// TIA Portal V19 export
FUNCTION_BLOCK "A0304_Manager_FB"   // FB94, LAD
TITLE = Manager A0304
// stored: MemoryReserve 100, SetENOAutomatically false
   VAR_INPUT
      AreaInterface : "AreaInterface";
      ZSI : "udt_ZoneSafetyInterface";
      DataIn : Struct
         PbScaricaPacco : Bool;
         PbReggiaturaConclusa : Bool;
         LsMatPres1Load : Bool;
         LsMatPres2Load : Bool;
         LsMatPres1UnLoad : Bool;
         LsMatPres2UnLoad : Bool;
      END_STRUCT;
      CIn : Struct
         Navetta : Struct
            Testa : Struct
               Ax : "Positioning_DOL_Machine_COut";
               PalettiEsterni : "ValveMachine_COut";
               PalettiInterni : "ValveMachine_COut";
            END_STRUCT;
            Coda : Struct
               Ax : "Positioning_DOL_Machine_COut";
               PalettiEsterni : "ValveMachine_COut";
               PalettiInterni : "ValveMachine_COut";
            END_STRUCT;
            Cumulativo : Struct
               PalettiEsterni : "ValveMachine_COut";
               PalettiInterni : "ValveMachine_COut";
            END_STRUCT;
            ReadyToRecive : Bool;
         END_STRUCT;
         Sollevamento : Struct
            ReadyToDrop : Bool;   // In posizione di deposito e pacco completato
         END_STRUCT;
         Antiribaltamento : Struct
            Work : Bool;
            Rest : Bool;
            PalettoPos0 : Bool;
         END_STRUCT;
         Manager03 : Struct
            IsWaiting_NoPiecesBefore : Bool;
         END_STRUCT;
         ProdManager : "Prod_Beam_Ctrl";
      END_STRUCT;
   END_VAR
   VAR_OUTPUT
      COut { ExternalAccessible := 'False'; ExternalVisible := 'False'; ExternalWritable := 'False'} : Struct
         Navetta : Struct
            EnableStopDoorOpeningReq : Bool;
            EnableStopInPhase : Bool;
            EnableStopProgrammed : Bool;
            Control_ON : Bool;
            CanMoveFreely : Bool;
            OP : Struct
               VAI_A_PRELIEVO : Bool;
               PRELIEVO : Bool;
               VAI_A_DEPOSITO : Bool;
               DEPOSITO : Bool;
            END_STRUCT;
         END_STRUCT;
         Sollevatore : Struct
            ReadyToRecive : Bool;
            OutOfWorkspace : Bool;
         END_STRUCT;
      END_STRUCT;
      MachineInterface : "MachineInterface";
   END_VAR
   VAR_IN_OUT
      Par_Navetta : Struct
         PosPrePrelievo : LReal;
         PosPrelievo : LReal;
         PosDeposito : LReal;
         ToleranceWindow : LReal;
      END_STRUCT;
   END_VAR
   VAR
      Alarm : Struct
         ShuttleNotEmpty : Bool;
         STOP_FineTurno : Bool;
         STOP_ControlloQualita : Bool;
         STOP_End_Of_Proroduction : Bool;
         TimeoutRimozionePaccoMES : Bool;
      END_STRUCT;
      Warning : Struct
         UnloadNotPossible : Bool;   // impossibile scaricare con le porte aperte
         TimeoutRimozionePaccoMES : Bool;
      END_STRUCT;
      OP_CND : Struct
         VaiAPrelievo : Array[0..15] of "OpCnd";
         Prelievo { S7_SetPoint := 'True'} : Array[0..15] of "OpCnd";
         VaiADeposito : Array[0..15] of "OpCnd";
         Deposito : Array[0..15] of "OpCnd";
      END_STRUCT;
      Sts : Struct
         SemiAut : Struct
            ON : Bool;
            PbMaterialFwd : Bool;
            Request : Bool;
         END_STRUCT;
         InPosDeposito : Bool;
         InPosPrePrelievo : Bool;
         InPosPrelievo : Bool;
         RichiestaVaiDeposito : Bool;
         RichiestaVaiPrelievo : Bool;
         IsStandstill : Bool;
         AlarmsPresence : Bool;
         WarningsPresence : Bool;
      END_STRUCT;
      Ctrl : Struct
         Cycle : Struct
            VaiAPrelievo : Bool;   // CICLO - Vai a Posizione di prelievo
            Prelievo : Bool;   // CICLO - Prelievo
            VaiADeposito : Bool;   // CICLO - Vai a Posizione di deposito
            Deposito : Bool;   // CICLO - Deposito
         END_STRUCT;
         ReggiaturaConclusa : Bool;
         ConfermaPaccoScaricato : Bool;
         Stop : Bool;
      END_STRUCT;
      AUX : Struct
         SemiAut_Pb : Bool;
         PbScaricaPacco : Bool;
         PbReggiaturaConclusa : Bool;
      END_STRUCT;
      TON_MatPres : IEC_TIMER;
      TON_Stop : IEC_TIMER;
      TON_ForceConfermaPaccoScraicato : IEC_TIMER;
      TON_TimeoutRimozionePaccoMES { S7_SetPoint := 'True'} : IEC_TIMER;
      TON_WngTimeoutRimozionePaccoMES { S7_SetPoint := 'True'} : IEC_TIMER;
      CycleWithShortPiece : Bool;
   END_VAR
   VAR_TEMP
      PE : Struct
         PbScaricaPacco : Bool;
         PbReggiaturaConclusa : Bool;
      END_STRUCT;
      Testa_InPosDeposito : Bool;
      Testa_InPosPrePrelievo : Bool;
      Testa_InPosPrelievo : Bool;
      Coda_InPosDeposito : Bool;
      Coda_InPosPrePrelievo : Bool;
      Coda_InPosPrelievo : Bool;
      ConteggioLayer_Navetta : Int;
      i : Int;
   END_VAR
   VAR CONSTANT
      OUTOFWORKSPACE : LReal := 1000.0;   // Quota fuori ingombro navetta con sollevatore
   END_VAR
   VAR_TEMP   // added for the SCL form of the ladder/FBD networks
      _w1 : Bool;
      _w2 : Bool;
      _w3 : Bool;
      _w4 : Bool;
      _w5 : Bool;
   END_VAR
BEGIN

REGION Network 1 (SCL): Reset Alarms
   IF #AreaInterface.RstAlarms THEN
       #Alarm.ShuttleNotEmpty := FALSE;
       #Warning.UnloadNotPossible:=FALSE;
       #Alarm.STOP_ControlloQualita := FALSE;
       #Alarm.STOP_End_Of_Proroduction := FALSE;
       #Alarm.STOP_FineTurno := FALSE;
       #Alarm.TimeoutRimozionePaccoMES := FALSE;
   END_IF;
END_REGION

REGION Network 2: PE
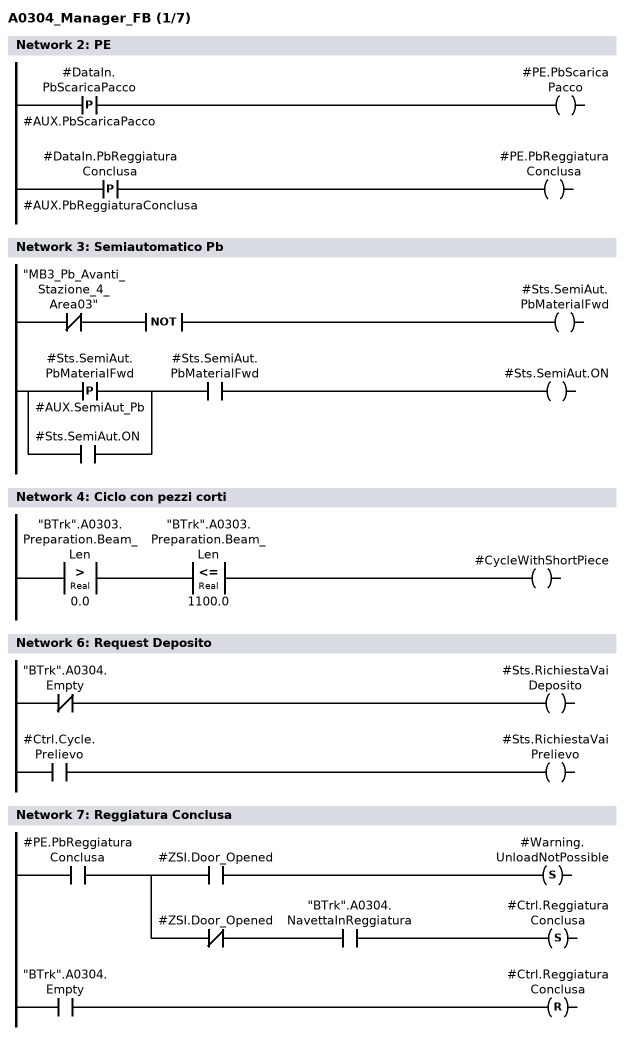
   RUNG wire#powerrail
      P_Contact(operand := #DataIn.PbScaricaPacco, bit := #AUX.PbScaricaPacco)
      Coil( #PE.PbScaricaPacco )
   END_RUNG
   RUNG wire#powerrail
      P_Contact(operand := #DataIn.PbReggiaturaConclusa, bit := #AUX.PbReggiaturaConclusa)
      Coil( #PE.PbReggiaturaConclusa )
   END_RUNG
   // the same network as SCL:
   #_w1 := #DataIn.PbScaricaPacco AND NOT #AUX.PbScaricaPacco;   // rising edge of #DataIn.PbScaricaPacco
   #AUX.PbScaricaPacco := #DataIn.PbScaricaPacco;
   #PE.PbScaricaPacco := #_w1;
   #_w2 := #DataIn.PbReggiaturaConclusa AND NOT #AUX.PbReggiaturaConclusa;   // rising edge of #DataIn.PbReggiaturaConclusa
   #AUX.PbReggiaturaConclusa := #DataIn.PbReggiaturaConclusa;
   #PE.PbReggiaturaConclusa := #_w2;
END_REGION

REGION Network 3: Semiautomatico Pb
   RUNG wire#powerrail
      I_Contact( "MB3_Pb_Avanti_Stazione_4_Area03" )
      Not()
      Coil( #Sts.SemiAut.PbMaterialFwd )
   END_RUNG
   RUNG wire#powerrail
      P_Contact(operand := #Sts.SemiAut.PbMaterialFwd, bit := #AUX.SemiAut_Pb)
      wire#w1
      Contact( #Sts.SemiAut.PbMaterialFwd )
      Coil( #Sts.SemiAut.ON )
   END_RUNG
   RUNG wire#powerrail
      Contact( #Sts.SemiAut.ON )
   END_RUNG wire#w1
   // the same network as SCL:
   #Sts.SemiAut.PbMaterialFwd := NOT (NOT "MB3_Pb_Avanti_Stazione_4_Area03");
   #_w1 := #Sts.SemiAut.PbMaterialFwd AND NOT #AUX.SemiAut_Pb;   // rising edge of #Sts.SemiAut.PbMaterialFwd
   #AUX.SemiAut_Pb := #Sts.SemiAut.PbMaterialFwd;
   #Sts.SemiAut.ON := (#_w1 OR #Sts.SemiAut.ON) AND #Sts.SemiAut.PbMaterialFwd;
END_REGION

REGION Network 4: Ciclo con pezzi corti
   RUNG wire#powerrail
      { S7_Templates := "SrcType := Real" } GT_Contact(in1 := "BTrk".A0303.Preparation.Beam_Len, in2 := 0.0)
      { S7_Templates := "SrcType := Real" } LE_Contact(in1 := "BTrk".A0303.Preparation.Beam_Len, in2 := 1100.0)
      Coil( #CycleWithShortPiece )
   END_RUNG
   // the same network as SCL:
   #CycleWithShortPiece := ("BTrk".A0303.Preparation.Beam_Len > 0.0) AND ("BTrk".A0303.Preparation.Beam_Len <= 1100.0);
END_REGION

REGION Network 6: Request Deposito
   RUNG wire#powerrail
      I_Contact( "BTrk".A0304.Empty )
      Coil( #Sts.RichiestaVaiDeposito )
   END_RUNG
   RUNG wire#powerrail
      Contact( #Ctrl.Cycle.Prelievo )
      Coil( #Sts.RichiestaVaiPrelievo )
   END_RUNG
   // the same network as SCL:
   #Sts.RichiestaVaiDeposito := NOT "BTrk".A0304.Empty;
   #Sts.RichiestaVaiPrelievo := #Ctrl.Cycle.Prelievo;
END_REGION

REGION Network 7: Reggiatura Conclusa
   RUNG wire#powerrail
      Contact( #PE.PbReggiaturaConclusa )
      wire#w1
      Contact( #ZSI.Door_Opened )
      S_Coil( #Warning.UnloadNotPossible )
   END_RUNG
   RUNG wire#w1
      I_Contact( #ZSI.Door_Opened )
      Contact( "BTrk".A0304.NavettaInReggiatura )
      S_Coil( #Ctrl.ReggiaturaConclusa )
   END_RUNG
   RUNG wire#powerrail
      Contact( "BTrk".A0304.Empty )
      R_Coil( #Ctrl.ReggiaturaConclusa )
   END_RUNG
   // the same network as SCL:
   IF #PE.PbReggiaturaConclusa AND #ZSI.Door_Opened THEN #Warning.UnloadNotPossible := TRUE; END_IF;
   IF #PE.PbReggiaturaConclusa AND NOT #ZSI.Door_Opened AND "BTrk".A0304.NavettaInReggiatura THEN
       #Ctrl.ReggiaturaConclusa := TRUE;
   END_IF;
   IF "BTrk".A0304.Empty THEN #Ctrl.ReggiaturaConclusa := FALSE; END_IF;
END_REGION

REGION Network 8: Conferma Pacco Scaricato
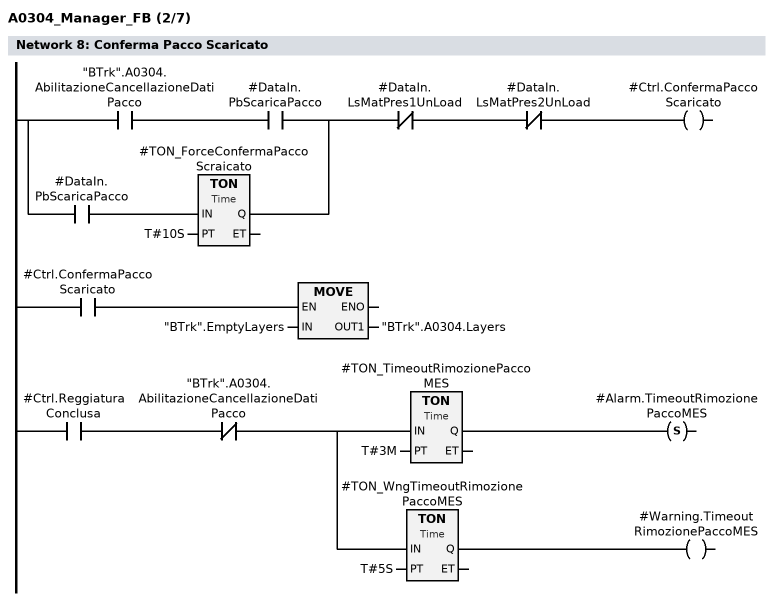
   RUNG wire#powerrail
      Contact( "BTrk".A0304.AbilitazioneCancellazioneDatiPacco )
      Contact( #DataIn.PbScaricaPacco )
      wire#w1
      I_Contact( #DataIn.LsMatPres1UnLoad )
      I_Contact( #DataIn.LsMatPres2UnLoad )
      Coil( #Ctrl.ConfermaPaccoScaricato )
   END_RUNG
   RUNG wire#powerrail
      Contact( #DataIn.PbScaricaPacco )
      { S7_Templates := "time_type := Time" } #TON_ForceConfermaPaccoScraicato.TON(pt := T#10S, et =>)
   END_RUNG wire#w1
   RUNG wire#powerrail
      Contact( #Ctrl.ConfermaPaccoScaricato )
      Move(in := "BTrk".EmptyLayers, out1 => "BTrk".A0304.Layers)
   END_RUNG
   RUNG wire#powerrail
      Contact( #Ctrl.ReggiaturaConclusa )
      I_Contact( "BTrk".A0304.AbilitazioneCancellazioneDatiPacco )
      wire#w2
      { S7_Templates := "time_type := Time" } #TON_TimeoutRimozionePaccoMES.TON(pt := T#3M, et =>)
      S_Coil( #Alarm.TimeoutRimozionePaccoMES )
   END_RUNG
   RUNG wire#w2
      { S7_Templates := "time_type := Time" } #TON_WngTimeoutRimozionePaccoMES.TON(pt := T#5S, et =>)
      Coil( #Warning.TimeoutRimozionePaccoMES )
   END_RUNG
   // the same network as SCL:
   #TON_ForceConfermaPaccoScraicato.TON(IN := #DataIn.PbScaricaPacco, PT := T#10S);
   #Ctrl.ConfermaPaccoScaricato := (("BTrk".A0304.AbilitazioneCancellazioneDatiPacco AND #DataIn.PbScaricaPacco) OR #TON_ForceConfermaPaccoScraicato.Q) AND NOT #DataIn.LsMatPres1UnLoad AND NOT #DataIn.LsMatPres2UnLoad;
   IF #Ctrl.ConfermaPaccoScaricato THEN "BTrk".A0304.Layers := "BTrk".EmptyLayers; END_IF;
   #_w1 := #Ctrl.ReggiaturaConclusa AND NOT "BTrk".A0304.AbilitazioneCancellazioneDatiPacco;
   #TON_TimeoutRimozionePaccoMES.TON(IN := #_w1, PT := T#3M);
   IF #TON_TimeoutRimozionePaccoMES.Q THEN #Alarm.TimeoutRimozionePaccoMES := TRUE; END_IF;
   #TON_WngTimeoutRimozionePaccoMES.TON(IN := #_w1, PT := T#5S);
   #Warning.TimeoutRimozionePaccoMES := #TON_WngTimeoutRimozionePaccoMES.Q;
END_REGION

REGION Network 10: Ax Navetta in posizione
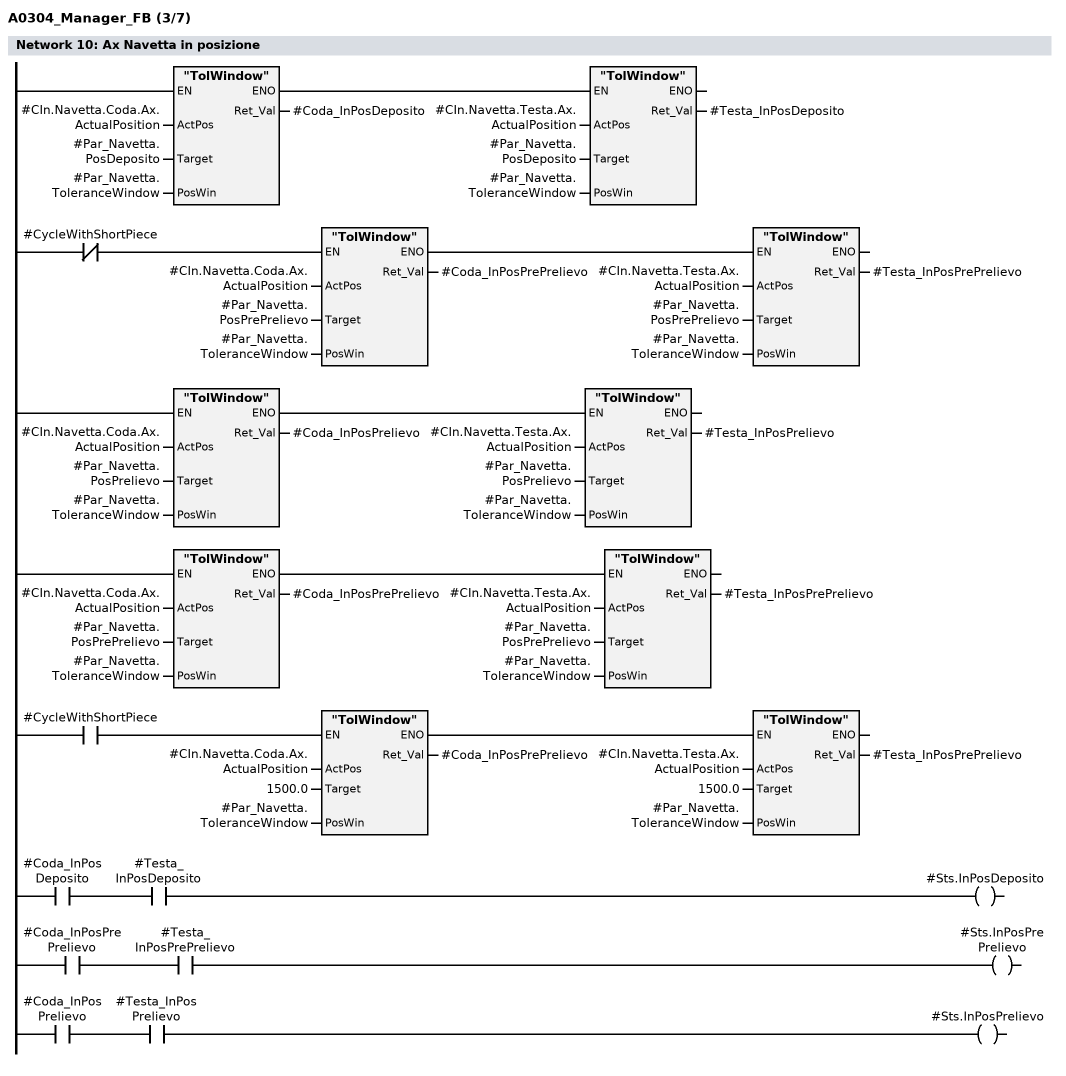
   RUNG wire#powerrail
      "TolWindow"(ActPos := #CIn.Navetta.Coda.Ax.ActualPosition, Target := #Par_Navetta.PosDeposito, PosWin := #Par_Navetta.ToleranceWindow, Ret_Val => #Coda_InPosDeposito)
      "TolWindow"(ActPos := #CIn.Navetta.Testa.Ax.ActualPosition, Target := #Par_Navetta.PosDeposito, PosWin := #Par_Navetta.ToleranceWindow, Ret_Val => #Testa_InPosDeposito)
   END_RUNG
   RUNG wire#powerrail
      I_Contact( #CycleWithShortPiece )
      "TolWindow"(ActPos := #CIn.Navetta.Coda.Ax.ActualPosition, Target := #Par_Navetta.PosPrePrelievo, PosWin := #Par_Navetta.ToleranceWindow, Ret_Val => #Coda_InPosPrePrelievo)
      "TolWindow"(ActPos := #CIn.Navetta.Testa.Ax.ActualPosition, Target := #Par_Navetta.PosPrePrelievo, PosWin := #Par_Navetta.ToleranceWindow, Ret_Val => #Testa_InPosPrePrelievo)
   END_RUNG
   RUNG wire#powerrail
      "TolWindow"(ActPos := #CIn.Navetta.Coda.Ax.ActualPosition, Target := #Par_Navetta.PosPrelievo, PosWin := #Par_Navetta.ToleranceWindow, Ret_Val => #Coda_InPosPrelievo)
      "TolWindow"(ActPos := #CIn.Navetta.Testa.Ax.ActualPosition, Target := #Par_Navetta.PosPrelievo, PosWin := #Par_Navetta.ToleranceWindow, Ret_Val => #Testa_InPosPrelievo)
   END_RUNG
   RUNG wire#powerrail
      "TolWindow"(ActPos := #CIn.Navetta.Coda.Ax.ActualPosition, Target := #Par_Navetta.PosPrePrelievo, PosWin := #Par_Navetta.ToleranceWindow, Ret_Val => #Coda_InPosPrePrelievo)
      "TolWindow"(ActPos := #CIn.Navetta.Testa.Ax.ActualPosition, Target := #Par_Navetta.PosPrePrelievo, PosWin := #Par_Navetta.ToleranceWindow, Ret_Val => #Testa_InPosPrePrelievo)
   END_RUNG
   RUNG wire#powerrail
      Contact( #CycleWithShortPiece )
      "TolWindow"(ActPos := #CIn.Navetta.Coda.Ax.ActualPosition, Target := 1500.0, PosWin := #Par_Navetta.ToleranceWindow, Ret_Val => #Coda_InPosPrePrelievo)
      "TolWindow"(ActPos := #CIn.Navetta.Testa.Ax.ActualPosition, Target := 1500.0, PosWin := #Par_Navetta.ToleranceWindow, Ret_Val => #Testa_InPosPrePrelievo)
   END_RUNG
   RUNG wire#powerrail
      Contact( #Coda_InPosDeposito )
      Contact( #Testa_InPosDeposito )
      Coil( #Sts.InPosDeposito )
   END_RUNG
   RUNG wire#powerrail
      Contact( #Coda_InPosPrePrelievo )
      Contact( #Testa_InPosPrePrelievo )
      Coil( #Sts.InPosPrePrelievo )
   END_RUNG
   RUNG wire#powerrail
      Contact( #Coda_InPosPrelievo )
      Contact( #Testa_InPosPrelievo )
      Coil( #Sts.InPosPrelievo )
   END_RUNG
   // the same network as SCL:
   #Coda_InPosDeposito := "TolWindow"(ActPos := #CIn.Navetta.Coda.Ax.ActualPosition,
                           Target := #Par_Navetta.PosDeposito,
                           PosWin := #Par_Navetta.ToleranceWindow,
                           ENO => #_w1);
   IF #_w1 THEN
       #Testa_InPosDeposito := "TolWindow"(ActPos := #CIn.Navetta.Testa.Ax.ActualPosition,
                               Target := #Par_Navetta.PosDeposito,
                               PosWin := #Par_Navetta.ToleranceWindow);
   END_IF;
   #Coda_InPosPrePrelievo := "TolWindow"(EN := NOT #CycleWithShortPiece,
                           ActPos := #CIn.Navetta.Coda.Ax.ActualPosition,
                           Target := #Par_Navetta.PosPrePrelievo,
                           PosWin := #Par_Navetta.ToleranceWindow,
                           ENO => #_w2);
   IF #_w2 THEN
       #Testa_InPosPrePrelievo := "TolWindow"(ActPos := #CIn.Navetta.Testa.Ax.ActualPosition,
                               Target := #Par_Navetta.PosPrePrelievo,
                               PosWin := #Par_Navetta.ToleranceWindow);
   END_IF;
   #Coda_InPosPrelievo := "TolWindow"(ActPos := #CIn.Navetta.Coda.Ax.ActualPosition,
                           Target := #Par_Navetta.PosPrelievo,
                           PosWin := #Par_Navetta.ToleranceWindow,
                           ENO => #_w3);
   IF #_w3 THEN
       #Testa_InPosPrelievo := "TolWindow"(ActPos := #CIn.Navetta.Testa.Ax.ActualPosition,
                               Target := #Par_Navetta.PosPrelievo,
                               PosWin := #Par_Navetta.ToleranceWindow);
   END_IF;
   #Coda_InPosPrePrelievo := "TolWindow"(ActPos := #CIn.Navetta.Coda.Ax.ActualPosition,
                           Target := #Par_Navetta.PosPrePrelievo,
                           PosWin := #Par_Navetta.ToleranceWindow,
                           ENO => #_w4);
   IF #_w4 THEN
       #Testa_InPosPrePrelievo := "TolWindow"(ActPos := #CIn.Navetta.Testa.Ax.ActualPosition,
                               Target := #Par_Navetta.PosPrePrelievo,
                               PosWin := #Par_Navetta.ToleranceWindow);
   END_IF;
   #Coda_InPosPrePrelievo := "TolWindow"(EN := #CycleWithShortPiece,
                           ActPos := #CIn.Navetta.Coda.Ax.ActualPosition,
                           Target := 1500.0,
                           PosWin := #Par_Navetta.ToleranceWindow,
                           ENO => #_w5);
   IF #_w5 THEN
       #Testa_InPosPrePrelievo := "TolWindow"(ActPos := #CIn.Navetta.Testa.Ax.ActualPosition,
                               Target := 1500.0,
                               PosWin := #Par_Navetta.ToleranceWindow);
   END_IF;
   #Sts.InPosDeposito := #Coda_InPosDeposito AND #Testa_InPosDeposito;
   #Sts.InPosPrePrelievo := #Coda_InPosPrePrelievo AND #Testa_InPosPrePrelievo;
   #Sts.InPosPrelievo := #Coda_InPosPrelievo AND #Testa_InPosPrelievo;
END_REGION

REGION Network 11: Ciclo Navetta
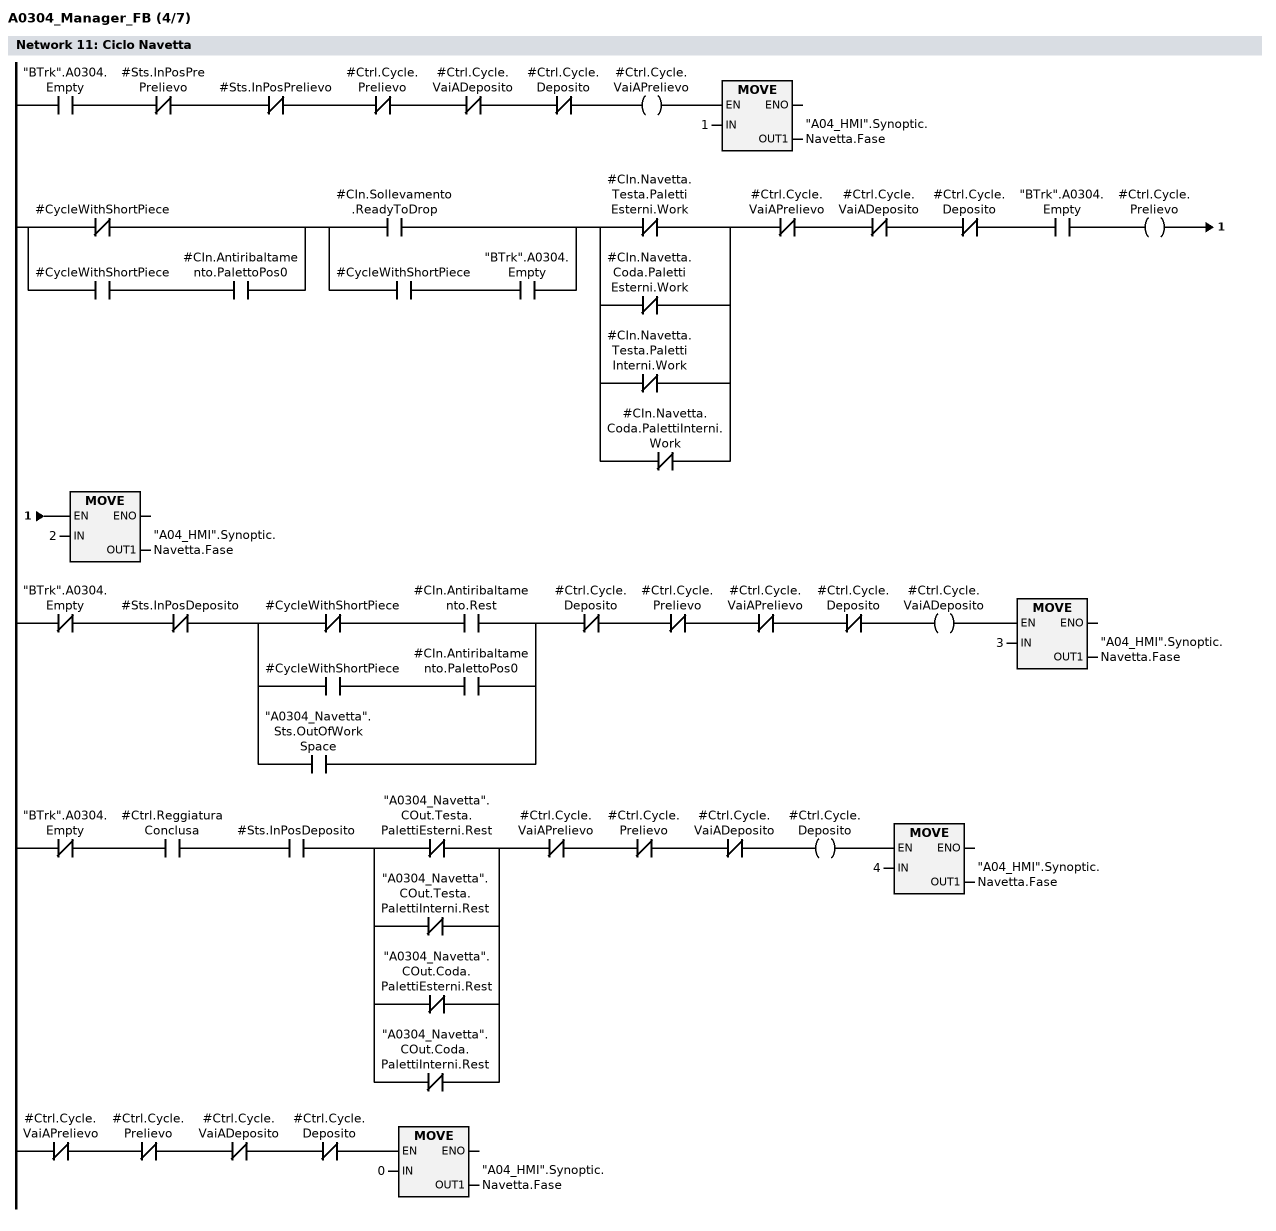
   RUNG wire#powerrail
      Contact( "BTrk".A0304.Empty )
      I_Contact( #Sts.InPosPrePrelievo )
      I_Contact( #Sts.InPosPrelievo )
      I_Contact( #Ctrl.Cycle.Prelievo )
      I_Contact( #Ctrl.Cycle.VaiADeposito )
      I_Contact( #Ctrl.Cycle.Deposito )
      Coil( #Ctrl.Cycle.VaiAPrelievo )
      Move(in := 1, out1 => "A04_HMI".Synoptic.Navetta.Fase)
   END_RUNG
   RUNG wire#powerrail
      I_Contact( #CycleWithShortPiece )
      wire#w1
      Contact( #CIn.Sollevamento.ReadyToDrop )
      wire#w2
      I_Contact( #CIn.Navetta.Testa.PalettiEsterni.Work )
      wire#w3
      I_Contact( #Ctrl.Cycle.VaiAPrelievo )
      I_Contact( #Ctrl.Cycle.VaiADeposito )
      I_Contact( #Ctrl.Cycle.Deposito )
      Contact( "BTrk".A0304.Empty )
      Coil( #Ctrl.Cycle.Prelievo )
      Move(in := 2, out1 => "A04_HMI".Synoptic.Navetta.Fase)
   END_RUNG
   RUNG wire#powerrail
      Contact( #CycleWithShortPiece )
      Contact( #CIn.Antiribaltamento.PalettoPos0 )
   END_RUNG wire#w1
   RUNG wire#w1
      Contact( #CycleWithShortPiece )
      Contact( "BTrk".A0304.Empty )
   END_RUNG wire#w2
   RUNG wire#w2
      I_Contact( #CIn.Navetta.Coda.PalettiEsterni.Work )
   END_RUNG wire#w3
   RUNG wire#w2
      I_Contact( #CIn.Navetta.Testa.PalettiInterni.Work )
   END_RUNG wire#w3
   RUNG wire#w2
      I_Contact( #CIn.Navetta.Coda.PalettiInterni.Work )
   END_RUNG wire#w3
   RUNG wire#powerrail
      I_Contact( "BTrk".A0304.Empty )
      I_Contact( #Sts.InPosDeposito )
      wire#w4
      I_Contact( #CycleWithShortPiece )
      Contact( #CIn.Antiribaltamento.Rest )
      wire#w5
      I_Contact( #Ctrl.Cycle.Deposito )
      I_Contact( #Ctrl.Cycle.Prelievo )
      I_Contact( #Ctrl.Cycle.VaiAPrelievo )
      I_Contact( #Ctrl.Cycle.Deposito )
      Coil( #Ctrl.Cycle.VaiADeposito )
      Move(in := 3, out1 => "A04_HMI".Synoptic.Navetta.Fase)
   END_RUNG
   RUNG wire#w4
      Contact( #CycleWithShortPiece )
      Contact( #CIn.Antiribaltamento.PalettoPos0 )
   END_RUNG wire#w5
   RUNG wire#w4
      Contact( "A0304_Navetta".Sts.OutOfWorkSpace )
   END_RUNG wire#w5
   RUNG wire#powerrail
      I_Contact( "BTrk".A0304.Empty )
      Contact( #Ctrl.ReggiaturaConclusa )
      Contact( #Sts.InPosDeposito )
      wire#w6
      I_Contact( "A0304_Navetta".COut.Testa.PalettiEsterni.Rest )
      wire#w7
      I_Contact( #Ctrl.Cycle.VaiAPrelievo )
      I_Contact( #Ctrl.Cycle.Prelievo )
      I_Contact( #Ctrl.Cycle.VaiADeposito )
      Coil( #Ctrl.Cycle.Deposito )
      Move(in := 4, out1 => "A04_HMI".Synoptic.Navetta.Fase)
   END_RUNG
   RUNG wire#w6
      I_Contact( "A0304_Navetta".COut.Testa.PalettiInterni.Rest )
   END_RUNG wire#w7
   RUNG wire#w6
      I_Contact( "A0304_Navetta".COut.Coda.PalettiEsterni.Rest )
   END_RUNG wire#w7
   RUNG wire#w6
      I_Contact( "A0304_Navetta".COut.Coda.PalettiInterni.Rest )
   END_RUNG wire#w7
   RUNG wire#powerrail
      I_Contact( #Ctrl.Cycle.VaiAPrelievo )
      I_Contact( #Ctrl.Cycle.Prelievo )
      I_Contact( #Ctrl.Cycle.VaiADeposito )
      I_Contact( #Ctrl.Cycle.Deposito )
      Move(in := 0, out1 => "A04_HMI".Synoptic.Navetta.Fase)
   END_RUNG
   // the same network as SCL:
   #Ctrl.Cycle.VaiAPrelievo := "BTrk".A0304.Empty AND NOT #Sts.InPosPrePrelievo AND NOT #Sts.InPosPrelievo AND NOT #Ctrl.Cycle.Prelievo AND NOT #Ctrl.Cycle.VaiADeposito AND NOT #Ctrl.Cycle.Deposito;
   IF #Ctrl.Cycle.VaiAPrelievo THEN "A04_HMI".Synoptic.Navetta.Fase := 1; END_IF;
   #Ctrl.Cycle.Prelievo := (NOT #CycleWithShortPiece OR (#CycleWithShortPiece AND #CIn.Antiribaltamento.PalettoPos0)) AND (#CIn.Sollevamento.ReadyToDrop OR (#CycleWithShortPiece AND "BTrk".A0304.Empty)) AND (NOT #CIn.Navetta.Testa.PalettiEsterni.Work OR NOT #CIn.Navetta.Coda.PalettiEsterni.Work OR NOT #CIn.Navetta.Testa.PalettiInterni.Work OR NOT #CIn.Navetta.Coda.PalettiInterni.Work) AND NOT #Ctrl.Cycle.VaiAPrelievo AND NOT #Ctrl.Cycle.VaiADeposito AND NOT #Ctrl.Cycle.Deposito AND "BTrk".A0304.Empty;
   IF #Ctrl.Cycle.Prelievo THEN "A04_HMI".Synoptic.Navetta.Fase := 2; END_IF;
   #Ctrl.Cycle.VaiADeposito := NOT "BTrk".A0304.Empty AND NOT #Sts.InPosDeposito AND ((NOT #CycleWithShortPiece AND #CIn.Antiribaltamento.Rest) OR (#CycleWithShortPiece AND #CIn.Antiribaltamento.PalettoPos0) OR "A0304_Navetta".Sts.OutOfWorkSpace) AND NOT #Ctrl.Cycle.Deposito AND NOT #Ctrl.Cycle.Prelievo AND NOT #Ctrl.Cycle.VaiAPrelievo AND NOT #Ctrl.Cycle.Deposito;
   IF #Ctrl.Cycle.VaiADeposito THEN "A04_HMI".Synoptic.Navetta.Fase := 3; END_IF;
   #Ctrl.Cycle.Deposito := NOT "BTrk".A0304.Empty AND #Ctrl.ReggiaturaConclusa AND #Sts.InPosDeposito AND (NOT "A0304_Navetta".COut.Testa.PalettiEsterni.Rest OR NOT "A0304_Navetta".COut.Testa.PalettiInterni.Rest OR NOT "A0304_Navetta".COut.Coda.PalettiEsterni.Rest OR NOT "A0304_Navetta".COut.Coda.PalettiInterni.Rest) AND NOT #Ctrl.Cycle.VaiAPrelievo AND NOT #Ctrl.Cycle.Prelievo AND NOT #Ctrl.Cycle.VaiADeposito;
   IF #Ctrl.Cycle.Deposito THEN "A04_HMI".Synoptic.Navetta.Fase := 4; END_IF;
   IF NOT #Ctrl.Cycle.VaiAPrelievo AND NOT #Ctrl.Cycle.Prelievo AND NOT #Ctrl.Cycle.VaiADeposito AND NOT #Ctrl.Cycle.Deposito THEN
       "A04_HMI".Synoptic.Navetta.Fase := 0;
   END_IF;
END_REGION

REGION Network 12: Stati Navetta (da gestire)
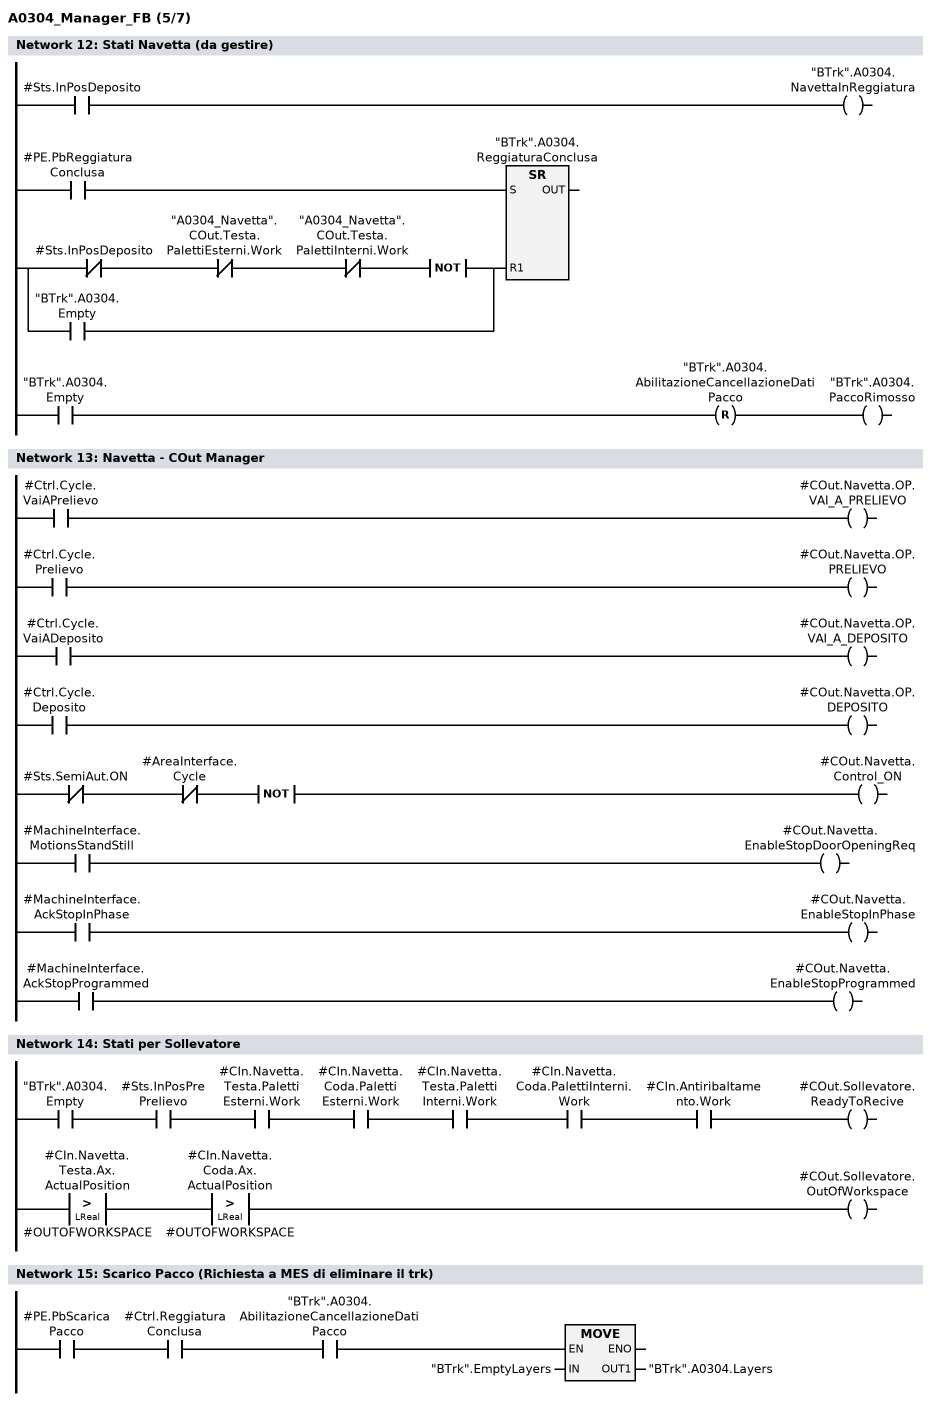
   RUNG wire#powerrail
      Contact( #Sts.InPosDeposito )
      Coil( "BTrk".A0304.NavettaInReggiatura )
   END_RUNG
   RUNG wire#powerrail
      Contact( #PE.PbReggiaturaConclusa )
      S_SR(operand := "BTrk".A0304.ReggiaturaConclusa, r1 := wire#w1)
   END_RUNG
   RUNG wire#powerrail
      I_Contact( #Sts.InPosDeposito )
      I_Contact( "A0304_Navetta".COut.Testa.PalettiEsterni.Work )
      I_Contact( "A0304_Navetta".COut.Testa.PalettiInterni.Work )
      Not()
   END_RUNG wire#w1
   RUNG wire#powerrail
      Contact( "BTrk".A0304.Empty )
   END_RUNG wire#w1
   RUNG wire#powerrail
      Contact( "BTrk".A0304.Empty )
      R_Coil( "BTrk".A0304.AbilitazioneCancellazioneDatiPacco )
      Coil( "BTrk".A0304.PaccoRimosso )
   END_RUNG
   // the same network as SCL:
   "BTrk".A0304.NavettaInReggiatura := #Sts.InPosDeposito;
   IF #PE.PbReggiaturaConclusa THEN
       "BTrk".A0304.ReggiaturaConclusa := TRUE;   // SR flip-flop
   END_IF;
   IF NOT (NOT #Sts.InPosDeposito AND NOT "A0304_Navetta".COut.Testa.PalettiEsterni.Work AND NOT "A0304_Navetta".COut.Testa.PalettiInterni.Work) OR "BTrk".A0304.Empty THEN
       "BTrk".A0304.ReggiaturaConclusa := FALSE;
   END_IF;
   IF "BTrk".A0304.Empty THEN "BTrk".A0304.AbilitazioneCancellazioneDatiPacco := FALSE; END_IF;
   "BTrk".A0304.PaccoRimosso := "BTrk".A0304.Empty;
END_REGION

REGION Network 13: Navetta - COut Manager
   RUNG wire#powerrail
      Contact( #Ctrl.Cycle.VaiAPrelievo )
      Coil( #COut.Navetta.OP.VAI_A_PRELIEVO )
   END_RUNG
   RUNG wire#powerrail
      Contact( #Ctrl.Cycle.Prelievo )
      Coil( #COut.Navetta.OP.PRELIEVO )
   END_RUNG
   RUNG wire#powerrail
      Contact( #Ctrl.Cycle.VaiADeposito )
      Coil( #COut.Navetta.OP.VAI_A_DEPOSITO )
   END_RUNG
   RUNG wire#powerrail
      Contact( #Ctrl.Cycle.Deposito )
      Coil( #COut.Navetta.OP.DEPOSITO )
   END_RUNG
   RUNG wire#powerrail
      I_Contact( #Sts.SemiAut.ON )
      I_Contact( #AreaInterface.Cycle )
      Not()
      Coil( #COut.Navetta.Control_ON )
   END_RUNG
   RUNG wire#powerrail
      Contact( #MachineInterface.MotionsStandStill )
      Coil( #COut.Navetta.EnableStopDoorOpeningReq )
   END_RUNG
   RUNG wire#powerrail
      Contact( #MachineInterface.AckStopInPhase )
      Coil( #COut.Navetta.EnableStopInPhase )
   END_RUNG
   RUNG wire#powerrail
      Contact( #MachineInterface.AckStopProgrammed )
      Coil( #COut.Navetta.EnableStopProgrammed )
   END_RUNG
   // the same network as SCL:
   #COut.Navetta.OP.VAI_A_PRELIEVO := #Ctrl.Cycle.VaiAPrelievo;
   #COut.Navetta.OP.PRELIEVO := #Ctrl.Cycle.Prelievo;
   #COut.Navetta.OP.VAI_A_DEPOSITO := #Ctrl.Cycle.VaiADeposito;
   #COut.Navetta.OP.DEPOSITO := #Ctrl.Cycle.Deposito;
   #COut.Navetta.Control_ON := NOT (NOT #Sts.SemiAut.ON AND NOT #AreaInterface.Cycle);
   #COut.Navetta.EnableStopDoorOpeningReq := #MachineInterface.MotionsStandStill;
   #COut.Navetta.EnableStopInPhase := #MachineInterface.AckStopInPhase;
   #COut.Navetta.EnableStopProgrammed := #MachineInterface.AckStopProgrammed;
END_REGION

REGION Network 14: Stati per Sollevatore
   RUNG wire#powerrail
      Contact( "BTrk".A0304.Empty )
      Contact( #Sts.InPosPrePrelievo )
      Contact( #CIn.Navetta.Testa.PalettiEsterni.Work )
      Contact( #CIn.Navetta.Coda.PalettiEsterni.Work )
      Contact( #CIn.Navetta.Testa.PalettiInterni.Work )
      Contact( #CIn.Navetta.Coda.PalettiInterni.Work )
      Contact( #CIn.Antiribaltamento.Work )
      Coil( #COut.Sollevatore.ReadyToRecive )
   END_RUNG
   RUNG wire#powerrail
      { S7_Templates := "SrcType := LReal" } GT_Contact(in1 := #CIn.Navetta.Testa.Ax.ActualPosition, in2 := #OUTOFWORKSPACE)
      { S7_Templates := "SrcType := LReal" } GT_Contact(in1 := #CIn.Navetta.Coda.Ax.ActualPosition, in2 := #OUTOFWORKSPACE)
      Coil( #COut.Sollevatore.OutOfWorkspace )
   END_RUNG
   // the same network as SCL:
   #COut.Sollevatore.ReadyToRecive := "BTrk".A0304.Empty AND #Sts.InPosPrePrelievo AND #CIn.Navetta.Testa.PalettiEsterni.Work AND #CIn.Navetta.Coda.PalettiEsterni.Work AND #CIn.Navetta.Testa.PalettiInterni.Work AND #CIn.Navetta.Coda.PalettiInterni.Work AND #CIn.Antiribaltamento.Work;
   #COut.Sollevatore.OutOfWorkspace := (#CIn.Navetta.Testa.Ax.ActualPosition > #OUTOFWORKSPACE) AND (#CIn.Navetta.Coda.Ax.ActualPosition > #OUTOFWORKSPACE);
END_REGION

REGION Network 15: Scarico Pacco (Richiesta a MES di eliminare il trk)
   RUNG wire#powerrail
      Contact( #PE.PbScaricaPacco )
      Contact( #Ctrl.ReggiaturaConclusa )
      Contact( "BTrk".A0304.AbilitazioneCancellazioneDatiPacco )
      Move(in := "BTrk".EmptyLayers, out1 => "BTrk".A0304.Layers)
   END_RUNG
   // the same network as SCL:
   IF #PE.PbScaricaPacco AND #Ctrl.ReggiaturaConclusa AND "BTrk".A0304.AbilitazioneCancellazioneDatiPacco THEN
       "BTrk".A0304.Layers := "BTrk".EmptyLayers;
   END_IF;
END_REGION

REGION Network 16 (SCL): Navetta completato / vuoto / conteggio pezzi
   // Conteggio Pezzi
   #ConteggioLayer_Navetta := 0;
   FOR #i := 1 TO "BTrk".A0304.BeamsPerLayer_Target DO
       IF "BTrk".A0304.Layers[#i].Layer[1].B_ID > 0 THEN
           #ConteggioLayer_Navetta += 1;
       END_IF;
   END_FOR;


   // pallet empty/full
   "BTrk".A0304.Empty := #ConteggioLayer_Navetta = 0;
   "BTrk".A0304.Layers_Qty := #ConteggioLayer_Navetta;
END_REGION

REGION Network 18: Allarme navetta non vuota
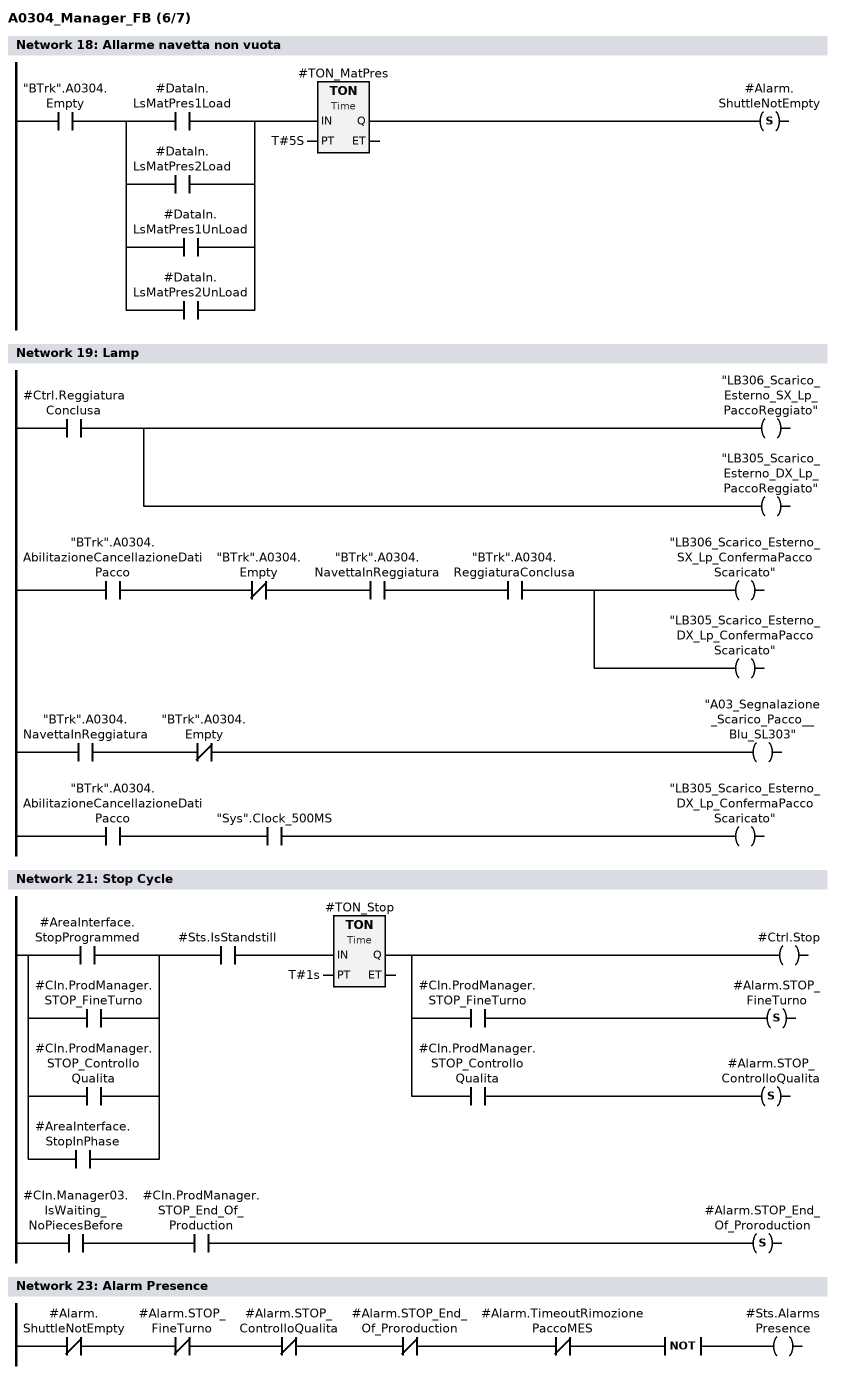
   RUNG wire#powerrail
      Contact( "BTrk".A0304.Empty )
      wire#w1
      Contact( #DataIn.LsMatPres1Load )
      wire#w2
      { S7_Templates := "time_type := Time" } #TON_MatPres.TON(pt := T#5S, et =>)
      S_Coil( #Alarm.ShuttleNotEmpty )
   END_RUNG
   RUNG wire#w1
      Contact( #DataIn.LsMatPres2Load )
   END_RUNG wire#w2
   RUNG wire#w1
      Contact( #DataIn.LsMatPres1UnLoad )
   END_RUNG wire#w2
   RUNG wire#w1
      Contact( #DataIn.LsMatPres2UnLoad )
   END_RUNG wire#w2
   // the same network as SCL:
   #TON_MatPres.TON(IN := "BTrk".A0304.Empty AND (#DataIn.LsMatPres1Load OR #DataIn.LsMatPres2Load OR #DataIn.LsMatPres1UnLoad OR #DataIn.LsMatPres2UnLoad),
                    PT := T#5S);
   IF #TON_MatPres.Q THEN #Alarm.ShuttleNotEmpty := TRUE; END_IF;
END_REGION

REGION Network 19: Lamp
   RUNG wire#powerrail
      Contact( #Ctrl.ReggiaturaConclusa )
      wire#w1
      Coil( "LB306_Scarico_Esterno_SX_Lp_PaccoReggiato" )
   END_RUNG
   RUNG wire#w1
      Coil( "LB305_Scarico_Esterno_DX_Lp_PaccoReggiato" )
   END_RUNG
   RUNG wire#powerrail
      Contact( "BTrk".A0304.AbilitazioneCancellazioneDatiPacco )
      I_Contact( "BTrk".A0304.Empty )
      Contact( "BTrk".A0304.NavettaInReggiatura )
      Contact( "BTrk".A0304.ReggiaturaConclusa )
      wire#w2
      Coil( "LB306_Scarico_Esterno_SX_Lp_ConfermaPaccoScaricato" )
   END_RUNG
   RUNG wire#w2
      Coil( "LB305_Scarico_Esterno_DX_Lp_ConfermaPaccoScaricato" )
   END_RUNG
   RUNG wire#powerrail
      Contact( "BTrk".A0304.NavettaInReggiatura )
      I_Contact( "BTrk".A0304.Empty )
      Coil( "A03_Segnalazione_Scarico_Pacco__Blu_SL303" )
   END_RUNG
   RUNG wire#powerrail
      Contact( "BTrk".A0304.AbilitazioneCancellazioneDatiPacco )
      Contact( "Sys".Clock_500MS )
      Coil( "LB305_Scarico_Esterno_DX_Lp_ConfermaPaccoScaricato" )
   END_RUNG
   // the same network as SCL:
   "LB306_Scarico_Esterno_SX_Lp_PaccoReggiato" := #Ctrl.ReggiaturaConclusa;
   "LB305_Scarico_Esterno_DX_Lp_PaccoReggiato" := #Ctrl.ReggiaturaConclusa;
   "LB306_Scarico_Esterno_SX_Lp_ConfermaPaccoScaricato" := "BTrk".A0304.AbilitazioneCancellazioneDatiPacco AND NOT "BTrk".A0304.Empty AND "BTrk".A0304.NavettaInReggiatura AND "BTrk".A0304.ReggiaturaConclusa;
   "LB305_Scarico_Esterno_DX_Lp_ConfermaPaccoScaricato" := "LB306_Scarico_Esterno_SX_Lp_ConfermaPaccoScaricato";
   "A03_Segnalazione_Scarico_Pacco__Blu_SL303" := "BTrk".A0304.NavettaInReggiatura AND NOT "BTrk".A0304.Empty;
   "LB305_Scarico_Esterno_DX_Lp_ConfermaPaccoScaricato" := "BTrk".A0304.AbilitazioneCancellazioneDatiPacco AND "Sys".Clock_500MS;
END_REGION

REGION Network 21: Stop Cycle
   RUNG wire#powerrail
      Contact( #AreaInterface.StopProgrammed )
      wire#w1
      Contact( #Sts.IsStandstill )
      { S7_Templates := "time_type := Time" } #TON_Stop.TON(pt := T#1s, et =>)
      wire#w2
      Coil( #Ctrl.Stop )
   END_RUNG
   RUNG wire#powerrail
      Contact( #CIn.ProdManager.STOP_FineTurno )
   END_RUNG wire#w1
   RUNG wire#powerrail
      Contact( #CIn.ProdManager.STOP_ControlloQualita )
   END_RUNG wire#w1
   RUNG wire#powerrail
      Contact( #AreaInterface.StopInPhase )
   END_RUNG wire#w1
   RUNG wire#w2
      Contact( #CIn.ProdManager.STOP_FineTurno )
      S_Coil( #Alarm.STOP_FineTurno )
   END_RUNG
   RUNG wire#w2
      Contact( #CIn.ProdManager.STOP_ControlloQualita )
      S_Coil( #Alarm.STOP_ControlloQualita )
   END_RUNG
   RUNG wire#powerrail
      Contact( #CIn.Manager03.IsWaiting_NoPiecesBefore )
      Contact( #CIn.ProdManager.STOP_End_Of_Production )
      S_Coil( #Alarm.STOP_End_Of_Proroduction )
   END_RUNG
   // the same network as SCL:
   #TON_Stop.TON(IN := (#AreaInterface.StopProgrammed OR #CIn.ProdManager.STOP_FineTurno OR #CIn.ProdManager.STOP_ControlloQualita OR #AreaInterface.StopInPhase) AND #Sts.IsStandstill,
                 PT := T#1s);
   #Ctrl.Stop := #TON_Stop.Q;
   IF #TON_Stop.Q AND #CIn.ProdManager.STOP_FineTurno THEN #Alarm.STOP_FineTurno := TRUE; END_IF;
   IF #TON_Stop.Q AND #CIn.ProdManager.STOP_ControlloQualita THEN
       #Alarm.STOP_ControlloQualita := TRUE;
   END_IF;
   IF #CIn.Manager03.IsWaiting_NoPiecesBefore AND #CIn.ProdManager.STOP_End_Of_Production THEN
       #Alarm.STOP_End_Of_Proroduction := TRUE;
   END_IF;
END_REGION

REGION Network 23: Alarm Presence
   RUNG wire#powerrail
      I_Contact( #Alarm.ShuttleNotEmpty )
      I_Contact( #Alarm.STOP_FineTurno )
      I_Contact( #Alarm.STOP_ControlloQualita )
      I_Contact( #Alarm.STOP_End_Of_Proroduction )
      I_Contact( #Alarm.TimeoutRimozionePaccoMES )
      Not()
      Coil( #Sts.AlarmsPresence )
   END_RUNG
   // the same network as SCL:
   #Sts.AlarmsPresence := NOT (NOT #Alarm.ShuttleNotEmpty AND NOT #Alarm.STOP_FineTurno AND NOT #Alarm.STOP_ControlloQualita AND NOT #Alarm.STOP_End_Of_Proroduction AND NOT #Alarm.TimeoutRimozionePaccoMES);
END_REGION

REGION Network 24: Warnings presence
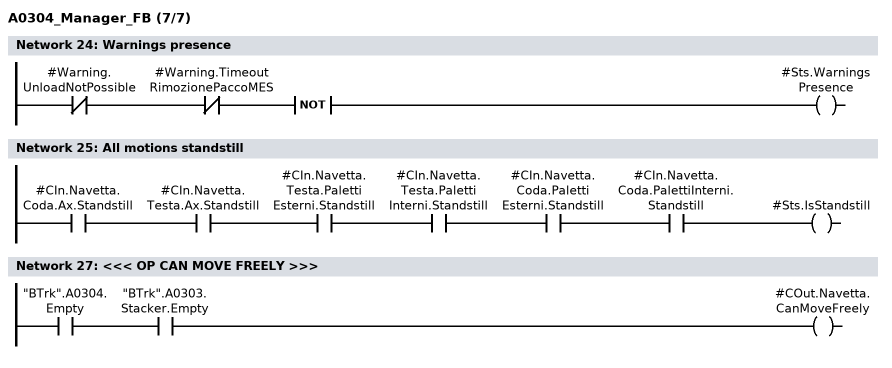
   RUNG wire#powerrail
      I_Contact( #Warning.UnloadNotPossible )
      I_Contact( #Warning.TimeoutRimozionePaccoMES )
      Not()
      Coil( #Sts.WarningsPresence )
   END_RUNG
   // the same network as SCL:
   #Sts.WarningsPresence := NOT (NOT #Warning.UnloadNotPossible AND NOT #Warning.TimeoutRimozionePaccoMES);
END_REGION

REGION Network 25: All motions standstill
   RUNG wire#powerrail
      Contact( #CIn.Navetta.Coda.Ax.Standstill )
      Contact( #CIn.Navetta.Testa.Ax.Standstill )
      Contact( #CIn.Navetta.Testa.PalettiEsterni.Standstill )
      Contact( #CIn.Navetta.Testa.PalettiInterni.Standstill )
      Contact( #CIn.Navetta.Coda.PalettiEsterni.Standstill )
      Contact( #CIn.Navetta.Coda.PalettiInterni.Standstill )
      Coil( #Sts.IsStandstill )
   END_RUNG
   // the same network as SCL:
   #Sts.IsStandstill := #CIn.Navetta.Coda.Ax.Standstill AND #CIn.Navetta.Testa.Ax.Standstill AND #CIn.Navetta.Testa.PalettiEsterni.Standstill AND #CIn.Navetta.Testa.PalettiInterni.Standstill AND #CIn.Navetta.Coda.PalettiEsterni.Standstill AND #CIn.Navetta.Coda.PalettiInterni.Standstill;
END_REGION

REGION Network 26 (SCL): Collect machine to area interface
   #MachineInterface.AlarmsPresence := #Sts.AlarmsPresence;

   #MachineInterface.WarningPresence := #Sts.WarningsPresence;

   #MachineInterface.MotionsStandStill := #Sts.IsStandstill;

   #MachineInterface.AutReady := #AreaInterface.Aut AND NOT #Sts.AlarmsPresence;


   #MachineInterface.AckStopInPhase := #AreaInterface.StopInPhase AND #Ctrl.Stop;

   #MachineInterface.AckStopProgrammed := #AreaInterface.StopProgrammed AND #Ctrl.Stop;


   #MachineInterface.Aborting := #AreaInterface.Aut AND #Sts.AlarmsPresence;
END_REGION

REGION Network 27: <<< OP CAN MOVE FREELY >>>
   RUNG wire#powerrail
      Contact( "BTrk".A0304.Empty )
      Contact( "BTrk".A0303.Stacker.Empty )
      Coil( #COut.Navetta.CanMoveFreely )
   END_RUNG
   // the same network as SCL:
   #COut.Navetta.CanMoveFreely := "BTrk".A0304.Empty AND "BTrk".A0303.Stacker.Empty;
END_REGION
END_FUNCTION_BLOCK
